{attribute 'pack_mode' := '1'}
TYPE ST_TrafficLightColorDataIn :
STRUCT
	sCellID						: STRING(30);
	sID							: STRING(30);

END_STRUCT
END_TYPE

(* stored: Version 1.1.0.1, ProductVersion 3.1.4024.5
   DUT ST_TrafficLightColorDataIn: Id {7a3a10de-0634-4867-856b-f6e139925a18} *)
